(* CODESYS project tc3_component.library
   Company: Zerlauth
   DefaultNamespace: Tc3_Component
   Version: 0.0.0.0
   Author: Peter Zerlauth
   DocFormat: reStructuredText
   Placeholder: Tc3_Component
   Description: ISA88 State Model with Observer and Events
   Title: Tc3_Component

Project tree, tasks and I/O mapping:
  libraries: Tc2_Standard, * (Beckhoff Automation GmbH); Tc2_System, * (Beckhoff Automation GmbH); Tc2_Utilities, * (Beckhoff Automation GmbH)
  Component/
    Event/
      data type E_Error
      data type E_Event
      function block FB_Event [ST]: FB_init, M_Abort, M_AddBOOL, M_AddINT, M_AddREAL, M_AddSTRING, M_AddTIME, M_Arguments, M_Complete, M_Debug, M_Default, M_Error, M_Hold, M_Information, M_Pause, M_Stop, M_Warning, P_Logger
      interface I_Event: M_Abort, M_AddBOOL, M_AddINT, M_AddREAL, M_AddSTRING, M_AddTIME, M_Complete, M_Debug, M_Error, M_Hold, M_Information, M_Pause, M_Stop, M_Warning, P_Logger
      data type ST_Event
      data type ST_EventFlags
    Info/
      function block FB_Info [ST]: FB_init, P_Class, P_Comment, P_Instance, P_Timestamp
      interface I_Info: P_Class, P_Comment, P_Instance, P_Timestamp
    Observer/
      function block FB_Observer [ST]: FB_exit, M_Attach, M_Clear, M_Detach, M_Find, M_Index, M_Notify, P_Length
      interface I_Observer: M_Attach, M_Detach, M_Notify
    Sequence/
      data type E_Sequence
      function block FB_Sequence [ST]: FB_init, M_Await, M_Reset, P_Number
      interface I_Sequence: M_Await, M_Reset, P_Number
    data type E_Mode
    data type E_Request
    data type E_State
    function block FB_Component [ST]: M_Mode, M_Request, M_Aborted, M_Aborting, M_Completed, M_Completing, M_Execute, M_Held, M_Holding, M_Idle, M_Initialise, M_Paused, M_Pausing, M_Resetting, M_Resuming, M_Running, M_Starting, M_Stopped, M_Stopping, M_Unholding, FB_init, M_Cycle, M_OnMode, M_OnNotify, M_OnState, P_Event, P_Identifier, P_Info, P_Mode, P_Observer, P_State
    interface I_Component: M_Cycle, M_Mode, M_OnNotify, M_Request, P_Event, P_Identifier, P_Info, P_Mode, P_Observer, P_State
  List/
    function block FB_ListComponent [ST]: FB_exit, M_Add, M_Clear, M_Find, M_Index, M_Remove, M_Request, P_Length
    function block FB_ListLogger [ST]: FB_exit, M_Add, M_Clear, M_Find, M_Index, M_Remove, P_Length
    function block FB_ListObject [ST]: FB_exit, M_Add, M_Clear, M_Find, M_Index, M_Remove, P_Length
    function block FB_ListString [ST]: FB_exit, M_Add, M_Clear, M_Find, M_Index, M_Remove, P_Length
    interface I_ListComponent: M_Add, M_Clear, M_Find, M_Index, M_Remove, M_Request, P_Length
    interface I_ListLogger: M_Add, M_Clear, M_Find, M_Index, M_Remove, P_Length
    interface I_ListObject: M_Add, M_Clear, M_Find, M_Index, M_Remove, P_Length
    interface I_ListString: M_Add, M_Clear, M_Find, M_Index, M_Remove, P_Length
  Logger/
    function block FB_FileLogger [ST]: M_Log
    function block FB_Logger [ST]: M_Log
    function block FB_TcLogger [ST]: M_Log
  LoggerFactory/
    function block FB_LoggerFactory [ST]: M_Attach, M_Dettach, M_Find, M_Log, M_Publish, M_Remove, M_Reset, M_Start, P_Tags
    interface I_Logger: M_Log
    data type ST_LoggerFactoryTags
  Module/
    function block FB_ModuleBase [ST]: M_Aborted, M_Attach, M_Cycle, M_Dettach, M_Idle, M_Initialise, M_OnMode, M_Resetting, M_Resuming, M_Running, M_Starting, M_Stopped, M_Unholding
    interface I_Module
  Object/
    interface I_Object
  Utils/
    Analog/
      function block AnalogInput [ST]: P_Identifier, P_State, P_Value
      function block AnalogInputREAL [ST]: P_Identifier, P_State, P_Value
      function block AnalogOutput [ST]: FB_init, P_Identifier, P_State, P_Value
      interface I_AnalogChannel: P_Value
    Digital/
      function block FB_DigitalInput [ST]: P_Identifier, P_State, P_Value
      function block FB_DigitalOutput [ST]: P_Identifier, P_State, P_Value
      interface I_Channel: P_Identifier, P_State
      interface I_DigitalChannel: P_Value
    File/
      function block FB_File [ST]: M_Append, M_AppendLine, M_Close, M_Create, M_Delete, M_Load, M_Open, M_Read, M_Write, P_Error
      interface I_File: M_Append, M_AppendLine, M_Close, M_Create, M_Delete, M_Load, M_Open, M_Read, M_Write, P_Error
    function block FB_Debounce [ST]
  global variables Globals
  Klassendiagramm
  global variables Parameters
*)

// Component/Event/E_Error
{attribute 'qualified_only'}
{attribute 'strict'}
{attribute 'to_string'}
TYPE E_Error :
(
	None		:= 0,
    Pause       := 4,	
    Hold      	:= 8,
	Complete	:= 16,	
	Stop		:= 32,
	Abort       := 64
);
END_TYPE

// Component/Event/E_Event
{attribute 'qualified_only'}
{attribute 'strict'}
{attribute 'to_string'}
TYPE E_Event :
(
	Verbose			:= 0,
	Debug			:= 1,
	Information		:= 2,
	Warning			:= 3,
	Error			:= 4
);
END_TYPE

// Component/Event/ST_Event
TYPE ST_Event :
STRUCT
	iSource:		I_Component;
	eEventType:		E_Event;
	nTimestamp:   	ULINT;
	sID:			STRING(10);
	sInstance:		STRING(255);
	sClass:			STRING(255);
	sMessage:		STRING(255);
	sDefault:		STRING(255);
	sArguments:		STRING(255);
	stFlags:		ST_EventFlags;
END_STRUCT
END_TYPE

// Component/Event/ST_EventFlags
TYPE ST_EventFlags :
STRUCT
	bActive:		BIT;
	bRemove:		BIT;
	bPause:			BIT;
	bHold:			BIT;
	bComplete:		BIT;
END_STRUCT
END_TYPE

// Component/Sequence/E_Sequence
{attribute 'qualified_only'}
{attribute 'strict'}
{attribute 'to_string'}
TYPE E_Sequence :
(
	Manual			:= -32768,
	Start			:= 0,
	Done			:= 32767
);
END_TYPE

// Component/E_Mode
{attribute 'qualified_only'}
{attribute 'strict'}
{attribute 'to_string'}
TYPE E_Mode :
(
	{attribute 'hide'}
    Undefined   := 0,
	Automatic   := 1,
    Semiauto    := 2,
	Manual		:= 3
);
END_TYPE

// Component/E_Request
{attribute 'qualified_only'}
{attribute 'strict'}
{attribute 'to_string'}
TYPE E_Request :
(
	{attribute 'hide'}
    Undefined   := 0,
	Reset       := 1,
    Start       := 2,
    Pause       := 4,	
    Hold      	:= 8,
	Complete	:= 16,	
	Stop		:= 32,
	Abort       := 64
);
END_TYPE

// Component/E_State
{attribute 'qualified_only'}
{attribute 'strict'}
{attribute 'to_string'}
TYPE E_State :
(
	{attribute 'hide'}
	Undefined		:= 0,
	Idle			:= 1,
	
// Start
	Starting		:= 2,
	Execute			:= 3,
	
// Pause
	Pausing			:= 4,
	Paused			:= 5,
	Resuming		:= 6,
	
// Hold
	Holding			:= 7,
	Held			:= 8,
	Unholding		:= 9,
	
// Complete
	Completing		:= 10,
	Completed		:= 11,

// Stop
	Stopping		:= 12,
	Stopped			:= 13,

// Abort	
	Aborting		:= 14,
	Aborted			:= 15,

// Reset
	Resetting		:= 16

);
END_TYPE

// LoggerFactory/ST_LoggerFactoryTags
TYPE ST_LoggerFactoryTags :
STRUCT
	bInformation:				BOOL;
	bWarning:					BOOL;
	bError:						BOOL;
	bPause:						BOOL;
	bHold:						BOOL;
	bComplete:					BOOL;	
END_STRUCT
END_TYPE

// Globals
VAR_GLOBAL
	{IF (defined (release))}
    	{attribute 'hide'}
	{END_IF}
	fbLogger:			FB_Logger;
END_VAR

// Parameters
{attribute 'qualified_only'}
VAR_GLOBAL CONSTANT
	nEvents:						INT:= 49;		// Maximum of Events displayed in each Module
END_VAR

// Component/Event/FB_Event
FUNCTION_BLOCK FB_Event IMPLEMENTS I_Event
VAR_INPUT
END_VAR
VAR_OUTPUT
END_VAR
VAR
	fbList:				FB_ListString;
	iParent:			I_Component;
	iLogger:			I_Logger;
	stEvent:			ST_Event;
END_VAR

// https://github.com/PeterZerlauth/Tc3_Component

METHOD FB_init : BOOL
VAR_INPUT
	bInitRetains : BOOL; // if TRUE, the retain variables are initialized (warm start / cold start)
	bInCopyCode : BOOL;  // if TRUE, the instance afterwards gets moved into the copy code (online change)
	iParent:			I_Component;
END_VAR
THIS^.iParent:= iParent;
END_METHOD

METHOD PUBLIC M_Abort
VAR_INPUT
	sMessage:				STRING(255);
	sID:					STRING(10);
END_VAR
stEvent.sMessage:= sMessage;
stEvent.iSource:= iParent;
stEvent.sInstance:= iParent.P_Info.P_Instance;
stEvent.sClass:= iParent.P_Info.P_Class;
stEvent.eEventType:= E_Event.Error;
stEvent.nTimestamp:= F_GetSystemTime();
stEvent.sID:= sID;
stEvent.sDefault:= M_Default(sMessage);
stEvent.sArguments:= M_Arguments();
stEvent.stFlags.bActive:= TRUE;
stEvent.stFlags.bRemove:= FALSE;
stEvent.stFlags.bPause:= FALSE;
stEvent.stFlags.bHold:= FALSE;
stEvent.stFlags.bComplete:= FALSE;

IF iLogger <> 0 THEN
	iLogger.M_Log(stEvent);
ELSE
	fbLogger.M_Log(stEvent);
END_IF

iParent.M_Request(E_Request.Abort);
END_METHOD

METHOD PUBLIC M_AddBOOL
VAR_INPUT
	Value: 	bool;
END_VAR
fbList.M_Add(BOOL_TO_STRING(Value));
END_METHOD

METHOD PUBLIC M_AddINT
VAR_INPUT
	Value: 	LINT;
END_VAR
fbList.M_Add(LINT_TO_STRING(Value));
END_METHOD

METHOD PUBLIC M_AddREAL
VAR_INPUT
	Value: 	Lreal;
	Decimals: INT;
END_VAR
fbList.M_Add(LREAL_TO_FMTSTR(Value, Decimals, TRUE));
END_METHOD

METHOD PUBLIC M_AddSTRING
VAR_INPUT
	Value: STRING(255);
END_VAR
fbList.M_Add(Value);
END_METHOD

METHOD PUBLIC M_AddTIME
VAR_INPUT
	Value: 	TIME;
END_VAR
fbList.M_Add(TIME_TO_STRING(Value));
END_METHOD

METHOD INTERNAL M_Arguments : STRING(255)
VAR_INPUT
END_VAR
VAR
	nIndex:			INT;
END_VAR
WHILE nIndex < fbList. P_Length DO
	M_Arguments:= Concat(Concat(M_Arguments, fbList.M_Index(nIndex)), '$N');
	nIndex:= nIndex + 1;
END_WHILE

fbList.M_Clear();
END_METHOD

METHOD PUBLIC M_Complete
VAR_INPUT
	sMessage:				STRING(255);
	sID:					STRING(10);
END_VAR
stEvent.sMessage:= sMessage;
stEvent.iSource:= iParent;
stEvent.sInstance:= iParent.P_Info.P_Instance;
stEvent.sClass:= iParent.P_Info.P_Class;
stEvent.eEventType:= E_Event.Error;
stEvent.nTimestamp:= F_GetSystemTime();
stEvent.sID:= sID;
stEvent.sDefault:= M_Default(sMessage);
stEvent.sArguments:= M_Arguments();
stEvent.stFlags.bActive:= TRUE;
stEvent.stFlags.bRemove:= FALSE;
stEvent.stFlags.bPause:= FALSE;
stEvent.stFlags.bHold:= False;
stEvent.stFlags.bComplete:= TRUE;

IF iLogger <> 0 THEN
	iLogger.M_Log(stEvent);
ELSE
	iParent.M_Request(E_Request.Complete);
	fbLogger.M_Log(stEvent);
END_IF
END_METHOD

METHOD PUBLIC M_Debug
VAR_INPUT
	Message:				STRING(255);
END_VAR
stEvent.sMessage:= Message;
stEvent.iSource:= iParent;
stEvent.sInstance:= iParent.P_Info.P_Instance;
stEvent.sClass:= iParent.P_Info.P_Class;
stEvent.eEventType:= E_Event.Debug;
stEvent.nTimestamp:= F_GetSystemTime();
stEvent.sID:= '';
stEvent.sDefault:= M_Default(Message);
stEvent.sArguments:= M_Arguments();
stEvent.stFlags.bActive:= TRUE;
stEvent.stFlags.bRemove:= TRUE;
stEvent.stFlags.bPause:= FALSE;
stEvent.stFlags.bHold:= FALSE;
stEvent.stFlags.bComplete:= FALSE;

IF iLogger <> 0 THEN
	iLogger.M_Log(stEvent);
ELSE
	fbLogger.M_Log(stEvent);
END_IF
END_METHOD

METHOD INTERNAL M_Default : STRING(255)
VAR_INPUT
	sMessage:		STRING(255);
END_VAR
VAR
	nIndex:		   	DINT;
	nPosition: 		INT;
END_VAR
nPosition:= Find(sMessage, '%s');
WHILE nPosition <> 0 DO
	sMessage:= Replace(sMessage, fbList.M_Index(nIndex), 2, nPosition);
	nPosition:= Find(sMessage, '%s');
	nIndex:= nIndex + 1;
END_WHILE
M_Default:= sMessage;
END_METHOD

METHOD PUBLIC M_Error
VAR_INPUT
	sMessage:				STRING(255);
	sID:					STRING(10);
END_VAR
stEvent.sMessage:= sMessage;
stEvent.iSource:= iParent;
stEvent.sInstance:= iParent.P_Info.P_Instance;
stEvent.sClass:= iParent.P_Info.P_Class;
stEvent.eEventType:= E_Event.Error;
stEvent.nTimestamp:= F_GetSystemTime();
stEvent.sID:= sID;
stEvent.sDefault:= M_Default(sMessage);
stEvent.sArguments:= M_Arguments();
stEvent.stFlags.bActive:= TRUE;
stEvent.stFlags.bRemove:= TRUE;
stEvent.stFlags.bPause:= FALSE;
stEvent.stFlags.bHold:= FALSE;
stEvent.stFlags.bComplete:= FALSE;

IF iLogger <> 0 THEN
	iLogger.M_Log(stEvent);
ELSE
	fbLogger.M_Log(stEvent);
END_IF
END_METHOD

METHOD PUBLIC M_Hold
VAR_INPUT
	sMessage:				STRING(255);
	sID:					STRING(10);
END_VAR
stEvent.sMessage:= sMessage;
stEvent.iSource:= iParent;
stEvent.sInstance:= iParent.P_Info.P_Instance;
stEvent.sClass:= iParent.P_Info.P_Class;
stEvent.eEventType:= E_Event.Error;
stEvent.nTimestamp:= F_GetSystemTime();
stEvent.sID:= sID;
stEvent.sDefault:= M_Default(sMessage);
stEvent.sArguments:= M_Arguments();
stEvent.stFlags.bActive:= TRUE;
stEvent.stFlags.bRemove:= FALSE;
stEvent.stFlags.bPause:= FALSE;
stEvent.stFlags.bHold:= TRUE;
stEvent.stFlags.bComplete:= FALSE;

IF iLogger <> 0 THEN
	iLogger.M_Log(stEvent);
ELSE
	iParent.M_Request(E_Request.Hold);
	fbLogger.M_Log(stEvent);
END_IF
END_METHOD

METHOD PUBLIC M_Information
VAR_INPUT
	Message:				STRING(255);
	ID:						STRING(10);
END_VAR
stEvent.sMessage:= Message;
stEvent.iSource:= iParent;
stEvent.sInstance:= iParent.P_Info.P_Instance;
stEvent.sClass:= iParent.P_Info.P_Class;
stEvent.eEventType:= E_Event.Information;
stEvent.nTimestamp:= F_GetSystemTime();
stEvent.sID:= ID;
stEvent.sDefault:= M_Default(Message);
stEvent.sArguments:= M_Arguments();
stEvent.stFlags.bActive:= TRUE;
stEvent.stFlags.bRemove:= TRUE;
stEvent.stFlags.bPause:= FALSE;
stEvent.stFlags.bHold:= FALSE;
stEvent.stFlags.bComplete:= FALSE;

IF iLogger <> 0 THEN
	iLogger.M_Log(stEvent);
ELSE
	fbLogger.M_Log(stEvent);
END_IF
END_METHOD

METHOD PUBLIC M_Pause
VAR_INPUT
	sMessage:				STRING(255);
	sID:					STRING(10);
END_VAR
stEvent.sMessage:= sMessage;
stEvent.iSource:= iParent;
stEvent.sInstance:= iParent.P_Info.P_Instance;
stEvent.sClass:= iParent.P_Info.P_Class;
stEvent.eEventType:= E_Event.Error;
stEvent.nTimestamp:= F_GetSystemTime();
stEvent.sID:= sID;
stEvent.sDefault:= M_Default(sMessage);
stEvent.sArguments:= M_Arguments();
stEvent.stFlags.bActive:= TRUE;
stEvent.stFlags.bRemove:= FALSE;
stEvent.stFlags.bPause:= TRUE;
stEvent.stFlags.bHold:= FALSE;
stEvent.stFlags.bComplete:= FALSE;

IF iLogger <> 0 THEN
	iLogger.M_Log(stEvent);
ELSE
	iParent.M_Request(E_Request.Pause);
	fbLogger.M_Log(stEvent);
END_IF
END_METHOD

METHOD PUBLIC M_Stop
VAR_INPUT
	sMessage:				STRING(255);
	sID:					STRING(10);
END_VAR
stEvent.sMessage:= sMessage;
stEvent.iSource:= iParent;
stEvent.sInstance:= iParent.P_Info.P_Instance;
stEvent.sClass:= iParent.P_Info.P_Class;
stEvent.eEventType:= E_Event.Error;
stEvent.nTimestamp:= F_GetSystemTime();
stEvent.sID:= sID;
stEvent.sDefault:= M_Default(sMessage);
stEvent.sArguments:= M_Arguments();
stEvent.stFlags.bActive:= TRUE;
stEvent.stFlags.bRemove:= FALSE;
stEvent.stFlags.bPause:= FALSE;
stEvent.stFlags.bHold:= FALSE;
stEvent.stFlags.bComplete:= FALSE;

IF iLogger <> 0 THEN
	iLogger.M_Log(stEvent);
ELSE
	fbLogger.M_Log(stEvent);
END_IF

iParent.M_Request(E_Request.Stop);
END_METHOD

METHOD PUBLIC M_Warning
VAR_INPUT
	Message:				STRING(255);
	ID:						STRING(10);
END_VAR
stEvent.sMessage:= Message;
stEvent.iSource:= iParent;
stEvent.sInstance:= iParent.P_Info.P_Instance;
stEvent.sClass:= iParent.P_Info.P_Class;
stEvent.eEventType:= E_Event.Warning;
stEvent.nTimestamp:= F_GetSystemTime();
stEvent.sID:= ID;
stEvent.sDefault:= M_Default(Message);
stEvent.sArguments:= M_Arguments();
stEvent.stFlags.bActive:= TRUE;
stEvent.stFlags.bRemove:= TRUE;
stEvent.stFlags.bPause:= FALSE;
stEvent.stFlags.bHold:= FALSE;
stEvent.stFlags.bComplete:= FALSE;

IF iLogger<> 0 THEN
	iLogger.M_Log(stEvent);
ELSE
	fbLogger.M_Log(stEvent);
END_IF
END_METHOD

PROPERTY PUBLIC P_Logger : I_Logger
GET
P_Logger:= iLogger;
END_GET
SET
iLogger:= P_Logger;
END_SET
END_PROPERTY

END_FUNCTION_BLOCK

// Component/Event/I_Event
INTERFACE I_Event EXTENDS I_Object

METHOD PUBLIC M_Abort
VAR_INPUT
	sMessage:				STRING(255);
	sID:					STRING(10);
END_VAR
END_METHOD

METHOD PUBLIC M_AddBOOL
VAR_INPUT
	Value: 	BOOL;
END_VAR
END_METHOD

METHOD PUBLIC M_AddINT
VAR_INPUT
	Value: 	LINT;
END_VAR
END_METHOD

METHOD PUBLIC M_AddREAL
VAR_INPUT
	Value: 	Lreal;
	Decimals: INT;
END_VAR
END_METHOD

METHOD PUBLIC M_AddSTRING
VAR_INPUT
	Value: STRING(255);
END_VAR
END_METHOD

METHOD PUBLIC M_AddTIME
VAR_INPUT
	Value: 	TIME;
END_VAR
END_METHOD

METHOD PUBLIC M_Complete
VAR_INPUT
	sMessage:				STRING(255);
	sID:					STRING(10);
END_VAR
END_METHOD

METHOD PUBLIC M_Debug
VAR_INPUT
	Message:				STRING(255);
END_VAR
END_METHOD

METHOD PUBLIC M_Error
VAR_INPUT
	sMessage:				STRING(255);
	sID:					STRING(10);
END_VAR
END_METHOD

METHOD PUBLIC M_Hold
VAR_INPUT
	sMessage:				STRING(255);
	sID:					STRING(10);
END_VAR
END_METHOD

METHOD PUBLIC M_Information
VAR_INPUT
	Message:				STRING(255);
	ID:						STRING(10);
END_VAR
END_METHOD

METHOD PUBLIC M_Pause
VAR_INPUT
	sMessage:				STRING(255);
	sID:					STRING(10);
END_VAR
END_METHOD

METHOD PUBLIC M_Stop
VAR_INPUT
	sMessage:				STRING(255);
	sID:					STRING(10);
END_VAR
END_METHOD

METHOD PUBLIC M_Warning
VAR_INPUT
	Message:				STRING(255);
	ID:						STRING(10);
END_VAR
END_METHOD

PROPERTY PUBLIC P_Logger : I_Logger
GET
END_GET
SET
END_SET
END_PROPERTY

END_INTERFACE

// Object/I_Object
INTERFACE I_Object EXTENDS __SYSTEM.IQueryInterface

END_INTERFACE

// LoggerFactory/I_Logger
INTERFACE I_Logger EXTENDS I_Object

METHOD PUBLIC M_Log
VAR_INPUT
	stEvent:		ST_Event;
END_VAR
END_METHOD

END_INTERFACE

// List/FB_ListString
{attribute 'no_explicit_call' := 'do not call this POU directly'} 
FUNCTION_BLOCK FB_ListString IMPLEMENTS I_ListString
VAR
	pList: 			POINTER TO STRING(255);
	nLength:		DINT;
	{IF (defined (release))}
    	{attribute 'hide'}
	{END_IF}
	aList:			POINTER TO POINTER TO ARRAY [0..49] OF STRING(255):=ADR(pList);
END_VAR

// https://github.com/PeterZerlauth/Tc3_Component

METHOD FB_exit : BOOL
VAR_INPUT
	bInCopyCode : BOOL; // if TRUE, the exit method is called for exiting an instance that is copied afterwards (online change).
END_VAR
M_Clear();
END_METHOD

METHOD PUBLIC M_Add : BOOL
VAR_INPUT
	Object: 	STRING(255);
END_VAR
VAR
	pOldList: 	POINTER TO STRING(255);
END_VAR
IF Object <> '' THEN
	// First Item
	IF pList = 0 THEN
		nLength:= nLength + 1;
		pList:= __NEW(STRING(255),DINT_TO_UDINT(nLength));
	ELSE
		// Item already in List
		IF M_Find(Object) = -1 THEN
			// backup 
			pOldList:= pList;
			// new Length
			nLength:= nLength + 1;
			// new pointer
			pList:= __NEW(STRING(255),DINT_TO_UDINT(nLength));
			// restore
			Memcpy(pList,pOldList, SIZEOF(STRING(255))*DINT_TO_UDINT(nLength -1));
			// delete old
			__DELETE(pOldList);
		ELSE
			M_Add:= FALSE;	
			RETURN;
		END_IF
	END_IF
	IF pList = 0 THEN
		RETURN;
	END_IF
	// add new Object
	pList[nLength-1]:= Object;
	M_Add:= TRUE;
ELSE
	M_Add:= FALSE;	
END_IF
END_METHOD

METHOD PUBLIC M_Clear : BOOL
IF pList <> 0 THEN
	nLength:= 0;
	__DELETE(pList);
END_IF
M_Clear:= True;
END_METHOD

METHOD PUBLIC M_Find : DINT
VAR_INPUT
	Object: 	STRING(255);
END_VAR
VAR
	nIndex: 	UINT;
END_VAR
// Object already in List
M_Find := -1;
WHILE nIndex < nLength DO
    IF (pList[nIndex] = Object) THEN
        M_Find := nIndex;
        RETURN;
    END_IF
	nIndex := nIndex + 1;
END_WHILE
END_METHOD

METHOD PUBLIC M_Index : STRING(255)
VAR_INPUT
	Index: 	DINT;
END_VAR
IF Index <= nLength THEN
	M_Index:= pList[Index];
ELSE
	M_Index:= '';
END_IF
END_METHOD

METHOD PUBLIC M_Remove : BOOL
VAR_INPUT
	Object: 	STRING(255);
END_VAR
VAR
	pOldList:			POINTER TO STRING(255);
	nPosition: 			DINT;
END_VAR
IF Object <> '' THEN
	// First Item
	IF nLength >= 0 THEN
		// Item already in List
		nPosition:= M_Find(Object);
		IF nPosition <> -1 THEN
			// backup 
			pOldList:= pList;
			// new Length
			nLength:= nLength -1;
			// new pointer
			pList:= __NEW(POINTER TO I_Object,DINT_TO_UDINT(nLength));
			// restore lower part
			Memcpy(pList,pOldList, SIZEOF(STRING(255)) * DINT_TO_UDINT(nPosition));
			//pList[nPosition]:= iObject;
			Memcpy(pList + (SIZEOF(STRING(255))*nPosition),pOldList + (SIZEOF(STRING(255))*(nPosition + 1)), SIZEOF(STRING(255)) * DINT_TO_UDINT(nLength - nPosition));
			// delete old
			__DELETE(pOldList);
		ELSE
			M_Remove:= FALSE;	
			RETURN;
		END_IF
	ELSE
		M_Remove:= FALSE;	
		RETURN;
	END_IF
	M_Remove:= TRUE;
ELSE
	M_Remove:= FALSE;	
END_IF
END_METHOD

PROPERTY PUBLIC P_Length : DINT
GET
P_Length:= nLength;
END_GET
END_PROPERTY

END_FUNCTION_BLOCK

// List/I_ListString
INTERFACE I_ListString EXTENDS I_Object

METHOD PUBLIC M_Add : BOOL
VAR_INPUT
	Object: 	STRING(255);
END_VAR
END_METHOD

METHOD PUBLIC M_Clear : BOOL
END_METHOD

METHOD PUBLIC M_Find : DINT
VAR_INPUT
	Object: 	STRING(255);
END_VAR
END_METHOD

METHOD PUBLIC M_Index : STRING(255)
VAR_INPUT
	Index: 	DINT;
END_VAR
END_METHOD

METHOD PUBLIC M_Remove : BOOL
VAR_INPUT
	Object: 	STRING(255);
END_VAR
END_METHOD

PROPERTY PUBLIC P_Length : DINT
GET
END_GET
END_PROPERTY

END_INTERFACE

// Component/I_Component
INTERFACE I_Component EXTENDS I_Object

METHOD PUBLIC M_Cycle
VAR_INPUT
END_VAR
END_METHOD

METHOD PUBLIC M_Mode : BOOL
VAR_INPUT
	eMode:		E_Mode;
END_VAR
END_METHOD

METHOD PUBLIC M_OnNotify
VAR_INPUT
	eRequest:					E_Request;
	eMode:						E_Mode;
END_VAR
END_METHOD

METHOD PUBLIC M_Request : BOOL
VAR_INPUT
	eRequest:	E_Request;
END_VAR
END_METHOD

PROPERTY PUBLIC P_Event : I_Event
GET
END_GET
END_PROPERTY

PROPERTY PUBLIC P_Identifier : STRING(25)
GET
END_GET
SET
END_SET
END_PROPERTY

PROPERTY PUBLIC P_Info : I_Info
GET
END_GET
END_PROPERTY

PROPERTY PUBLIC P_Mode : E_Mode
GET
END_GET
END_PROPERTY

PROPERTY PUBLIC P_Observer : I_Observer
GET
END_GET
END_PROPERTY

PROPERTY PUBLIC P_State : E_State
GET
END_GET
END_PROPERTY

END_INTERFACE

// Component/Info/I_Info
INTERFACE I_Info EXTENDS I_Object

PROPERTY PUBLIC P_Class : String(255)
GET
END_GET
END_PROPERTY

PROPERTY PUBLIC P_Comment : String(255)
GET
END_GET
END_PROPERTY

PROPERTY PUBLIC P_Instance : String(255)
GET
END_GET
END_PROPERTY

PROPERTY PUBLIC P_Timestamp : ULINT
GET
END_GET
END_PROPERTY

END_INTERFACE

// Component/Observer/I_Observer
INTERFACE I_Observer

METHOD M_Attach : BOOL
VAR_INPUT
	Object: 	I_Component;
END_VAR
END_METHOD

METHOD M_Detach : BOOL
VAR_INPUT
	Object: 	I_Component;
END_VAR
END_METHOD

METHOD M_Notify : BOOL
VAR_INPUT
	eRequest:					E_Request;
	eMode:						E_Mode;
END_VAR
END_METHOD

END_INTERFACE

// Component/Info/FB_Info
FUNCTION_BLOCK PUBLIC FB_Info IMPLEMENTS I_Info
VAR_INPUT
	sIdentifier:						STRING(25);					// Identifier
END_VAR
VAR_OUTPUT
END_VAR
VAR
    sInstancePath:				REFERENCE TO STRING(255);
	fbReadSymInfo: 				PLC_ReadSymInfoByNameEx;
END_VAR
VAR_STAT
	nCycle: 					UDINT;
	nTimestamp: 				ULINT;
END_VAR

// https://github.com/PeterZerlauth/Tc3_Component
IF nCycle <> TwinCAT_SystemInfoVarList._TaskInfo[GETCURTASKINDEXEX()].CycleCount THEN
	nCycle:= TwinCAT_SystemInfoVarList._TaskInfo[GETCURTASKINDEXEX()].CycleCount;
	nTimestamp:= F_GetSystemTime();
END_IF

fbReadSymInfo(
	NETID:= , 
	PORT:= , 
	SYMNAME:= , 
	START:= , 
	TMOUT:= , 
	BUSY=> , 
	ERR=> , 
	ERRID=> , 
	SYMINFO=> , 
	OVTYPE=> , 
	OVCOMMENT=> );

METHOD FB_init : BOOL
VAR_INPUT
	bInitRetains : BOOL; // if TRUE, the retain variables are initialized (warm start / cold start)
	bInCopyCode : BOOL;  // if TRUE, the instance afterwards gets moved into the copy code (online change)
	sInstancePath:			REFERENCE TO STRING(255);
END_VAR
VAR
    sName:				STRING(255);
    nPosition:			INT;
END_VAR
THIS^.sInstancePath REF= sInstancePath;

sName := CONCAT(TwinCAT_SystemInfoVarList._AppInfo.ProjectName, '.');

nPosition := FIND(sInstancePath, sName);
IF nPosition > 0 THEN
    fbReadSymInfo.SYMNAME:= DELETE(sInstancePath, nPosition-1 + LEN(sName), 1);
END_IF

nPosition := FIND(fbReadSymInfo.SYMNAME, sName);

IF nPosition > 0 THEN
    fbReadSymInfo.SYMNAME:= DELETE(fbReadSymInfo.SYMNAME, nPosition - 1 + LEN(sName), 1);
END_IF

fbReadSymInfo.PORT:= TwinCAT_SystemInfoVarList._AppInfo.AdsPort;
fbReadSymInfo.START:= TRUE;
END_METHOD

PROPERTY PUBLIC P_Class : String(255)
GET
P_Class:= fbReadSymInfo.SYMINFO.symDataType;
END_GET
END_PROPERTY

PROPERTY PUBLIC P_Comment : String(255)
GET
P_Comment:= fbReadSymInfo.SYMINFO.symComment;
END_GET
END_PROPERTY

PROPERTY PUBLIC P_Instance : String(255)
GET
P_Instance:= fbReadSymInfo.SYMNAME;
END_GET
END_PROPERTY

PROPERTY PUBLIC P_Timestamp : ULINT
GET
P_Timestamp:= nTimestamp;
END_GET
END_PROPERTY

END_FUNCTION_BLOCK

// Component/Observer/FB_Observer
{attribute 'no_explicit_call'} 
FUNCTION_BLOCK PUBLIC FB_Observer IMPLEMENTS I_Observer
VAR
	pList: 			POINTER TO I_Component;
	nLength:		DINT;
	{attribute 'conditionalshow'}
	aList:			POINTER TO POINTER TO ARRAY [0..100] OF I_Component:=ADR(pList);
END_VAR

// https://github.com/PeterZerlauth/Tc3_Component

METHOD FB_exit : BOOL
VAR_INPUT
	bInCopyCode : BOOL; // if TRUE, the exit method is called for exiting an instance that is copied afterwards (online change).
END_VAR
M_Clear();
END_METHOD

METHOD M_Attach : BOOL
VAR_INPUT
	Object: 	I_Component;
END_VAR
VAR
	pOldList: 	POINTER TO I_Component;
END_VAR
IF Object <> 0 THEN
	// First Item
	IF pList = 0 THEN
		nLength:= nLength + 1;
		pList:= __NEW(POINTER TO I_Component,DINT_TO_UDINT(nLength));
	ELSE
		// Item already in List
		IF M_Find(Object) = -1 THEN
			// backup 
			pOldList:= pList;
			// new Length
			nLength:= nLength + 1;
			// new pointer
			pList:= __NEW(POINTER TO I_Component,DINT_TO_UDINT(nLength));
			// restore
			Memcpy(pList,pOldList, SIZEOF(POINTER TO I_Component)*DINT_TO_UDINT(nLength -1));
			// delete old
			__DELETE(pOldList);
		ELSE
			M_Attach:= FALSE;	
			RETURN;
		END_IF
	END_IF
	IF pList = 0 THEN
		RETURN;
	END_IF
	// add new Object
	pList[nLength-1]:= Object;
	M_Attach:= TRUE;
ELSE
	M_Attach:= FALSE;	
END_IF
END_METHOD

METHOD M_Clear
IF pList <> 0 THEN
	nLength:= 0;
	__DELETE(pList);
END_IF
END_METHOD

METHOD M_Detach : BOOL
VAR_INPUT
	Object: 	I_Component;
END_VAR
VAR
	pOldList:			POINTER TO I_Component;
	nPosition: 			DINT;
END_VAR
IF Object <> 0 THEN
	// First Item
	IF nLength >= 0 THEN
		// Item already in List
		nPosition:= M_Find(Object);
		IF nPosition <> -1 THEN
			// backup 
			pOldList:= pList;
			// new Length
			nLength:= nLength -1;
			// new pointer
			pList:= __NEW(POINTER TO I_Component,DINT_TO_UDINT(nLength));
			// restore lower part
			Memcpy(pList,pOldList, SIZEOF(POINTER TO I_Component) * DINT_TO_UDINT(nPosition));
			//pList[nPosition]:= iObject;
			Memcpy(pList + (SIZEOF(POINTER TO I_Component)*nPosition),pOldList + (SIZEOF(POINTER TO I_Component)*(nPosition + 1)), SIZEOF(POINTER TO I_Component) * DINT_TO_UDINT(nLength - nPosition));
			// delete old
			__DELETE(pOldList);
		ELSE
			M_Detach:= FALSE;	
			RETURN;
		END_IF
	ELSE
		M_Detach:= FALSE;	
		RETURN;
	END_IF
	M_Detach:= TRUE;
ELSE
	M_Detach:= FALSE;	
END_IF
END_METHOD

METHOD M_Find : DINT
VAR_INPUT
	Object: 	I_Component;
END_VAR
VAR
	nIndex: 	UINT;
END_VAR
// Object already in List
M_Find := -1;
WHILE nIndex < nLength DO
    IF (pList[nIndex] = Object) THEN
        M_Find := nIndex;
        RETURN;
    END_IF
	nIndex := nIndex + 1;
END_WHILE
END_METHOD

METHOD M_Index : I_Component
VAR_INPUT
	Index: 	DINT;
END_VAR
IF Index <= nLength THEN
	M_Index:= pList[Index];
END_IF
END_METHOD

METHOD M_Notify : BOOL
VAR_INPUT
	eRequest:					E_Request;
	eMode:						E_Mode;
END_VAR

VAR
	nIndex: 	INT;
END_VAR
WHILE nIndex < nLength DO
	pList[nIndex].M_OnNotify(eRequest, eMode);
	nIndex:= nIndex + 1; 
END_WHILE
END_METHOD

PROPERTY P_Length : DINT
GET
P_Length:= nLength;
END_GET
END_PROPERTY

END_FUNCTION_BLOCK

// Component/Sequence/FB_Sequence
FUNCTION_BLOCK FB_Sequence IMPLEMENTS I_Sequence
VAR_INPUT
END_VAR
VAR_OUTPUT
	sMessage:				STRING(255);
	nNumber:				INT;
END_VAR
VAR
	iParent:			I_Component;
	fbTimeout:			TON;
	fbDelay: 			TON;
END_VAR

// https://github.com/PeterZerlauth/Tc3_Component
IF iParent.P_Mode = E_Mode.Manual THEN
	nNumber:= E_Sequence.Manual;
END_IF

METHOD FB_init : BOOL
VAR_INPUT
	bInitRetains : BOOL; // if TRUE, the retain variables are initialized (warm start / cold start)
	bInCopyCode : BOOL;  // if TRUE, the instance afterwards gets moved into the copy code (online change)
	iParent:			I_Component;
END_VAR
THIS^.iParent:= iParent;
END_METHOD

METHOD PUBLIC M_Await 
VAR_INPUT
	sMessage:				STRING(255);		
	tTimeout:				TIME;
	tDelay:					TIME;	
	bPause:					BOOL;
	bReturn:				BOOL;
	nNumber:				INT;
END_VAR
THIS^.sMessage:= sMessage;
IF bReturn THEN
	IF tDelay <> T#0S THEN
		fbDelay(IN:= TRUE);
		IF fbDelay.Q THEN
			THIS^.nNumber:= nNumber;
			fbDelay(IN:= FALSE);
			IF bPause THEN
				IF iParent.P_Mode = E_Mode.Semiauto THEN
					iParent.M_Request(E_Request.Pause);		
				END_IF
			END_IF	
		END_IF
	ELSE
		THIS^.nNumber:= nNumber;
		fbTimeout(IN:= FALSE);
		IF bPause THEN
			IF iParent.P_Mode = E_Mode.Semiauto THEN
				iParent.M_Request(E_Request.Pause);		
			END_IF
		END_IF	
	END_IF		
ELSE
	IF tTimeout <> T#0S THEN
		fbTimeout(IN:= TRUE);
		IF fbTimeout.Q THEN
			iParent.P_Event.M_AddINT(THIS^.nNumber);
			iParent.P_Event.M_Stop('Timeout in sequence number %s', '');
		END_IF
	END_IF
END_IF
END_METHOD

METHOD M_Reset
nNumber:= E_Sequence.Start;
fbDelay(IN:= FALSE);
fbTimeout(IN:= FALSE);
END_METHOD

PROPERTY PUBLIC P_Number : int
GET
P_Number:= nNumber;
END_GET
SET
nNumber:= P_Number;
END_SET
END_PROPERTY

END_FUNCTION_BLOCK

// Component/Sequence/I_Sequence
INTERFACE I_Sequence EXTENDS I_Object

METHOD PUBLIC M_Await 
VAR_INPUT
	sMessage:				STRING(255);
	tTimeout:				TIME;
	tDelay:					TIME;	
	bPause:					BOOL;
	bReturn:				BOOL;
	nNumber:				INT;
END_VAR
END_METHOD

METHOD M_Reset
END_METHOD

PROPERTY PUBLIC P_Number : int
GET
END_GET
SET
END_SET
END_PROPERTY

END_INTERFACE

// Component/FB_Component
{attribute 'reflection'} 
{attribute 'no_explicit_call' := 'do not call this POU directly'} 
FUNCTION_BLOCK FB_Component IMPLEMENTS I_Component
VAR_INPUT
END_VAR
VAR_OUTPUT
END_VAR
VAR
    {attribute 'hide'}
	{attribute 'instance-path'} 
    {attribute 'noinit'}
    sInstancePath:					STRING(255);				// Instance-Path
	fbInfo:							FB_Info(sInstancePath);		// Info about function block
	fbObserver:						FB_Observer;				// Observer
	fbEvent:						FB_Event(THIS^);			// Event creator
	fbSequence:						FB_Sequence(THIS^);			// Sequence (abort = reset)
	eStateRequest:					E_Request;					// State command
	{attribute 'OPC.UA.DA' := '1'}
	{ attribute 'TcHmiSymbol' }
	eState:							E_State;					// Current state
    {attribute 'hide'}
	eStatePrevious:					E_State;					// Previous state
	eModeRequest:					E_Mode;						// Requested mode
	{attribute 'OPC.UA.DA' := '1'}
	{attribute 'TcHmiSymbol' }
	eMode:							E_Mode;						// Current mode
    {attribute 'hide'}
	eModePrevious:					E_Mode;						// Previous mode	
END_VAR

// https://github.com/PeterZerlauth/Tc3_Component

METHOD PUBLIC M_Mode : BOOL
VAR_INPUT
	eMode:		E_Mode;
END_VAR
IF eMode = E_Mode.Undefined THEN
	M_Mode:= TRUE;
ELSE
	IF THIS^.eMode = eMode THEN
		M_Mode:= TRUE;
	ELSE
		eModeRequest:= eMode;	
	END_IF	
END_IF
END_METHOD

METHOD PUBLIC M_Request : BOOL
VAR_INPUT
	eRequest:	E_Request;
END_VAR
// Request component states / Command Pattern
CASE eRequest OF
	E_Request.Undefined:
		M_Request:= TRUE;
		
	E_Request.Start:
		IF eState = E_State.Execute THEN
			M_Request:= TRUE;
		ELSE
			eStateRequest:= eRequest;				
		END_IF
		
	E_Request.Pause:
		IF eState >= E_State.Paused THEN
			M_Request:= TRUE;
		ELSE
			IF eStateRequest < eRequest THEN
				eStateRequest:= eRequest;				
			END_IF		
		END_IF
		
	E_Request.Hold:
		IF eState >= E_State.Held THEN
			M_Request:= TRUE;
		ELSE
			IF eStateRequest < eRequest THEN
				eStateRequest:= eRequest;				
			END_IF		
		END_IF
		
	E_Request.Complete:
		IF eState = E_State.Completed THEN
			M_Request:= TRUE;
		ELSE
			IF eStateRequest < eRequest THEN
				eStateRequest:= eRequest;				
			END_IF		
		END_IF
		
	E_Request.Stop:
		IF eState = E_State.Stopped THEN
			M_Request:= TRUE;
		ELSE
			IF eStateRequest < eRequest THEN
				eStateRequest:= eRequest;				
			END_IF		
		END_IF
		
	E_Request.Abort:
		IF eState = E_State.Aborted THEN
			M_Request:= TRUE;
		ELSE
			IF eStateRequest < eRequest THEN
				eStateRequest:= eRequest;				
			END_IF		
		END_IF

	E_Request.Reset:
		IF eState = E_State.Idle THEN
			M_Request:= TRUE;
		ELSE
			eStateRequest:= eRequest;			
		END_IF
END_CASE
END_METHOD

METHOD PROTECTED M_Aborted
VAR_INPUT
END_VAR
END_METHOD

METHOD PROTECTED M_Aborting : BOOL // Return state complete
VAR_INPUT
END_VAR
// State Aborting
M_Aborting:= TRUE;
END_METHOD

METHOD PROTECTED M_Completed
VAR_INPUT
END_VAR
END_METHOD

METHOD PROTECTED M_Completing : BOOL // Return state complete
VAR_INPUT
END_VAR
// State Completing
M_Completing:= True;
END_METHOD

METHOD PROTECTED M_Execute : BOOL // Return state complete
VAR_INPUT
END_VAR
M_Execute:= True;
END_METHOD

METHOD PROTECTED M_Held
VAR_INPUT
END_VAR
END_METHOD

METHOD PROTECTED M_Holding : BOOL // Return state complete
VAR_INPUT
END_VAR
// State Holding
M_Holding:= True;
END_METHOD

METHOD PROTECTED M_Idle
VAR_INPUT
END_VAR
// State Idle
END_METHOD

METHOD PROTECTED M_Initialise
VAR_INPUT
END_VAR
END_METHOD

METHOD PROTECTED M_Paused // Return state complete
VAR_INPUT
END_VAR
END_METHOD

METHOD PROTECTED M_Pausing : BOOL
VAR_INPUT
END_VAR
// State Holding
M_Pausing:= True;
END_METHOD

METHOD PROTECTED M_Resetting : BOOL // Return state complete
VAR_INPUT
END_VAR
// State Resetting
M_Resetting:= True;
END_METHOD

METHOD PROTECTED M_Resuming : BOOL // Return state complete
VAR_INPUT
END_VAR
// State Holding
M_Resuming:= True;
END_METHOD

METHOD PROTECTED M_Running
VAR_INPUT
END_VAR
// Will be called in all running states, for monitorings which not only in one state active
END_METHOD

METHOD PROTECTED M_Starting : BOOL // Return state complete
VAR_INPUT
END_VAR
// State Starting
M_Starting:= True;
END_METHOD

METHOD PROTECTED M_Stopped
VAR_INPUT
END_VAR
END_METHOD

METHOD PROTECTED M_Stopping : BOOL // Return state complete
VAR_INPUT
END_VAR
// State Stopping
M_Stopping:= True;
END_METHOD

METHOD PROTECTED M_Unholding : BOOL // Return state complete
VAR_INPUT
END_VAR
// State Holding
M_Unholding:= True;
END_METHOD

METHOD FB_init : BOOL
VAR_INPUT
	bInitRetains : BOOL; // if TRUE, the retain variables are initialized (warm start / cold start)
	bInCopyCode : BOOL:= TRUE;
END_VAR
M_Initialise();
END_METHOD

METHOD PUBLIC M_Cycle
VAR_INPUT
END_VAR
fbInfo();
fbObserver();
fbEvent();
fbSequence();

// Handle Module Type Package states
CASE eState OF
	E_State.Undefined:
		M_Initialise();
		eMode:= E_Mode.Automatic;
		eState:= E_State.Idle;					
		
	E_State.Resetting:
		M_Running();
		IF M_Resetting() THEN
			eState:= E_State.Idle;
			eStateRequest:= E_Request.Undefined;
		END_IF
		CASE eStateRequest OF
			E_Request.Stop:
				eState:= E_State.Stopping;
				
			E_Request.Abort:
				eState:= E_State.Aborting;
				
		END_CASE
		
	E_State.Idle:
		M_Running();
		M_Idle();
		CASE eStateRequest OF
			
			E_Request.Start:
				eState:= E_State.Starting;
				
			E_Request.Stop:
				eState:= E_State.Stopping;
				
			E_Request.Abort:
				eState:= E_State.Aborting;
				
			ELSE
				eStateRequest:= E_Request.Undefined;
				
		END_CASE

	E_State.Starting:
		M_Running();
		IF M_Starting() THEN
			eState:= E_State.Execute;
			eStateRequest:= E_Request.Undefined;
		END_IF
		CASE eStateRequest OF
			
			E_Request.Stop:
				eState:= E_State.Stopping;
				
			E_Request.Abort:
				eState:= E_State.Aborting;
				
		END_CASE

	E_State.Execute:
		M_Running();
		IF M_Execute() THEN
			CASE eStateRequest OF
				
				E_Request.Complete:
					eState:= E_State.Completing;
					
			END_CASE
		END_IF
		CASE eStateRequest OF
			E_Request.Complete:;
			E_Request.Stop:
				eState:= E_State.Stopping;
				
			E_Request.Abort:
				eState:= E_State.Aborting;

			E_Request.Hold:
				eState:= E_State.Holding;
				
			E_Request.Pause:
				eState:= E_State.Pausing;
				
			ELSE
				eStateRequest:= E_Request.Undefined;
				
		END_CASE
		
	E_State.Stopping:
		M_Running();
		IF M_Stopping() THEN
			eState:= E_State.Stopped;
			eStateRequest:= E_Request.Undefined;
		END_IF
		CASE eStateRequest OF
			
			E_Request.Abort:
				eState:= E_State.Aborting;
				
		END_CASE

	E_State.Stopped:
		M_Stopped();
		CASE eStateRequest OF
			
			E_Request.Abort:
				eState:= E_State.Aborting;
				
			E_Request.Reset:
				eState:= E_State.Resetting;
				
		ELSE
			eStateRequest:= E_Request.Undefined;				
		END_CASE
		
		
	E_State.Aborting:
		fbSequence.M_Reset();
		IF M_Aborting() THEN
			eState:= E_State.Aborted;
			eStateRequest:= E_Request.Undefined;
		END_IF
		
	E_State.Aborted:
		M_Aborted();
		CASE eStateRequest OF
			
			E_Request.Reset:
				eState:= E_State.Resetting;
				
		ELSE
			eStateRequest:= E_Request.Undefined;				
		END_CASE

		
	E_State.Pausing:
		M_Running();
		IF M_Pausing() THEN
			eState:= E_State.Paused;
			eStateRequest:= E_Request.Undefined;
		END_IF
		CASE eStateRequest OF
			
			E_Request.Stop:
				eState:= E_State.Stopping;
				
			E_Request.Abort:
				eState:= E_State.Aborting;

		END_CASE
		
	
	E_State.Paused:
		M_Running();
		M_Paused();
		CASE eStateRequest OF
			
			E_Request.Start:
				eState:= E_State.Resuming;
				
			E_Request.Stop:
				eState:= E_State.Stopping;
				
			E_Request.Abort:
				eState:= E_State.Aborting;
						
		ELSE
			eStateRequest:= E_Request.Undefined;

		END_CASE
		
	E_State.Resuming:
		M_Running();
		IF M_Resuming() THEN
			eState:= E_State.Execute;
		END_IF
		CASE eStateRequest OF
			
			E_Request.Stop:
				eState:= E_State.Stopping;
				
			E_Request.Abort:
				eState:= E_State.Aborting;

		END_CASE

	E_State.Holding:
		M_Running();
		IF M_Holding() THEN
			eState:= E_State.Held;
			eStateRequest:= E_Request.Undefined;
		END_IF
		CASE eStateRequest OF
			
			E_Request.Stop:
				eState:= E_State.Stopping;
				
			E_Request.Abort:
				eState:= E_State.Aborting;

		END_CASE

	E_State.Held:
		M_Running();
		M_Held();
		CASE eStateRequest OF
			
			E_Request.Start:
				eState:= E_State.Unholding;

			E_Request.Stop:
				eState:= E_State.Stopping;
				
			E_Request.Abort:
				eState:= E_State.Aborting;
				
			ELSE
				eStateRequest:= E_Request.Undefined;

		END_CASE
		
	E_State.Unholding:
		M_Running();
		IF M_Unholding() THEN
			eState:= E_State.Execute;
		END_IF
		CASE eStateRequest OF
			
			E_Request.Stop:
				eState:= E_State.Stopping;
				
			E_Request.Abort:
				eState:= E_State.Aborting;

		END_CASE
		
	E_State.Completing:
		M_Running();
		IF M_Completing() THEN
			eState:= E_State.Completed;
			eStateRequest:= E_Request.Undefined;
		END_IF
		CASE eStateRequest OF
			
			E_Request.Stop:
				eState:= E_State.Stopping;
				
			E_Request.Abort:
				eState:= E_State.Aborting;

		END_CASE
		
	E_State.Completed:
		M_Running();
		M_Completed();
		CASE eStateRequest OF
			
			E_Request.Stop:
				eState:= E_State.Stopping;
				
			E_Request.Abort:
				eState:= E_State.Aborting;
					
			E_Request.Reset:
				eState:= E_State.Resetting;
				
			ELSE
				eStateRequest:= E_Request.Undefined;
				
		END_CASE
		
END_CASE

IF eModeRequest <> E_Mode.Undefined THEN
	IF 	eMode <> eModeRequest THEN
		eMode:= eModeRequest;
		fbObserver.M_Notify(0, eMode);		
	END_IF
END_IF
eModeRequest:= E_Mode.Undefined;

// Detect mode changed
IF eModePrevious <> eMode THEN
	M_OnMode(eMode, eModePrevious);
	eModePrevious:= eMode;
END_IF
	
// Detect state changed
IF eStatePrevious <> eState THEN
	M_OnState(eState, eStatePrevious);
	eStatePrevious:= eState;
END_IF

CASE eStateRequest of
	E_Request.Undefined, E_Request.Start, E_Request.Pause, E_Request.Hold:
		// Ignore
	ELSE
		fbObserver.M_Notify(eStateRequest, 0);
END_CASE
END_METHOD

METHOD PROTECTED M_OnMode
VAR_INPUT
	eMode:							E_Mode;						// Current mode
	eModePrevious:					E_Mode;						// Previous mode	
END_VAR
END_METHOD

METHOD PUBLIC M_OnNotify
VAR_INPUT
	eRequest:					E_Request;
	eMode:						E_Mode;
END_VAR
// Method will be called by the Observer
M_Request(eRequest);
M_Mode(eMode);
END_METHOD

METHOD Protected M_OnState
VAR_INPUT
	eState:							E_State;						// Current state
	eStatePrevious:					E_State;						// Previous state	
END_VAR
END_METHOD

PROPERTY PUBLIC P_Event : I_Event
GET
P_Event:= fbEvent;
END_GET
END_PROPERTY

PROPERTY PUBLIC P_Identifier : STRING(25)
GET
P_Identifier:= fbInfo.sIdentifier;
END_GET
SET
PUBLIC 
VAR
END_VAR
fbInfo.sIdentifier:= P_Identifier;
END_SET
END_PROPERTY

PROPERTY PUBLIC P_Info : I_Info
GET
P_Info:= fbInfo;
END_GET
END_PROPERTY

PROPERTY PUBLIC P_Mode : E_Mode
GET
P_Mode:= eMode;
END_GET
END_PROPERTY

PROPERTY PUBLIC P_Observer : I_Observer
GET
P_Observer:= fbObserver;
END_GET
END_PROPERTY

PROPERTY PUBLIC P_State : E_State
GET
P_State:= eState;
END_GET
END_PROPERTY

END_FUNCTION_BLOCK

// List/FB_ListComponent
{attribute 'no_explicit_call' := 'do not call this POU directly'} 
FUNCTION_BLOCK FB_ListComponent IMPLEMENTS I_ListComponent
VAR
	nLength:		DINT;
	pList: 			POINTER TO I_Component;
	{IF (defined (release))}
    	{attribute 'hide'}
	{END_IF}
	aList:			POINTER TO POINTER TO ARRAY [0..49] OF I_Component:=ADR(pList);
END_VAR

// https://github.com/PeterZerlauth/Tc3_Component

METHOD FB_exit : BOOL
VAR_INPUT
	bInCopyCode : BOOL; // if TRUE, the exit method is called for exiting an instance that is copied afterwards (online change).
END_VAR
M_Clear();
END_METHOD

METHOD PUBLIC M_Add : BOOL
VAR_INPUT
	Object: 	I_Component;
END_VAR
VAR
	pOldList: 	POINTER TO I_Component;
END_VAR
IF Object <> 0 THEN
	// First Item
	IF pList = 0 THEN
		nLength:= nLength + 1;
		pList:= __NEW(POINTER TO I_Component,DINT_TO_UDINT(nLength));
	ELSE
		// Item already in List
		IF M_Find(Object) = -1 THEN
			// backup 
			pOldList:= pList;
			// new Length
			nLength:= nLength + 1;
			// new pointer
			pList:= __NEW(POINTER TO I_Component,DINT_TO_UDINT(nLength));
			// restore
			Memcpy(pList,pOldList, SIZEOF(POINTER TO I_Component)*DINT_TO_UDINT(nLength -1));
			// delete old
			__DELETE(pOldList);
		ELSE
			M_Add:= FALSE;	
			RETURN;
		END_IF
	END_IF
	IF pList = 0 THEN
		RETURN;
	END_IF
	// add new Object
	pList[nLength-1]:= Object;
	M_Add:= TRUE;
ELSE
	M_Add:= FALSE;	
END_IF
END_METHOD

METHOD PUBLIC M_Clear : BOOL
// Clear
IF pList <> 0 THEN
	nLength:= 0;
	__DELETE(pList);
END_IF
M_Clear:= TRUE;
END_METHOD

METHOD PUBLIC M_Find : DINT
VAR_INPUT
	Object: 	I_Component;
END_VAR
VAR
	nIndex: 	UINT;
END_VAR
// Find
M_Find := -1;
WHILE nIndex < nLength DO
    IF (pList[nIndex] = Object) THEN
        M_Find := nIndex;
        RETURN;
    END_IF
	nIndex := nIndex + 1;
END_WHILE
END_METHOD

METHOD PUBLIC M_Index : I_Component
VAR_INPUT
	Index: 	DINT;
END_VAR
// Index
IF Index <= nLength THEN
	M_Index:= pList[Index];
END_IF
END_METHOD

METHOD PUBLIC M_Remove : BOOL
VAR_INPUT
	Object: 	I_Component;
END_VAR
VAR
	pOldList:			POINTER TO I_Component;
	nPosition: 			DINT;
END_VAR
// Remove
IF Object <> 0 THEN
	// First Item
	IF nLength >= 0 THEN
		// Item already in List
		nPosition:= M_Find(Object);
		IF nPosition <> -1 THEN
			// backup 
			pOldList:= pList;
			// new Length
			nLength:= nLength -1;
			// new pointer
			pList:= __NEW(POINTER TO I_Component,DINT_TO_UDINT(nLength));
			// restore lower part
			Memcpy(pList,pOldList, SIZEOF(POINTER TO I_Object) * DINT_TO_UDINT(nPosition));
			//pList[nPosition]:= iObject;
			Memcpy(pList + (SIZEOF(POINTER TO I_Component)*nPosition),pOldList + (SIZEOF(POINTER TO I_Component)*(nPosition + 1)), SIZEOF(POINTER TO I_Component) * DINT_TO_UDINT(nLength - nPosition));
			// delete old
			__DELETE(pOldList);
		ELSE
			M_Remove:= FALSE;	
			RETURN;
		END_IF
	ELSE
		M_Remove:= FALSE;	
		RETURN;
	END_IF
	M_Remove:= TRUE;
ELSE
	M_Remove:= FALSE;	
END_IF
END_METHOD

METHOD PUBLIC M_Request : BOOL
VAR_INPUT
	eRequest:		E_Request;
END_VAR

VAR
	nIndex: 		INT;
END_VAR
M_Request:= TRUE;
WHILE nIndex < nLength DO
	M_Request:= M_Request AND M_Index(nIndex).M_Request(eRequest);
	nIndex:= nIndex +1;
END_WHILE
END_METHOD

PROPERTY PUBLIC P_Length : DINT
GET
P_Length:= nLength;
END_GET
END_PROPERTY

END_FUNCTION_BLOCK

// List/I_ListComponent
INTERFACE I_ListComponent

METHOD PUBLIC M_Add : BOOL
VAR_INPUT
	Object: 	I_Component;
END_VAR
END_METHOD

METHOD PUBLIC M_Clear : BOOL
END_METHOD

METHOD PUBLIC M_Find : DINT
VAR_INPUT
	Object: 	I_Component;
END_VAR
END_METHOD

METHOD PUBLIC M_Index : I_Component
VAR_INPUT
	Index: 	DINT;
END_VAR
END_METHOD

METHOD PUBLIC M_Remove : BOOL
VAR_INPUT
	Object: 	I_Component;
END_VAR
END_METHOD

METHOD PUBLIC M_Request : BOOL
VAR_INPUT
	eRequest:	E_Request;
END_VAR
END_METHOD

PROPERTY P_Length : DINT
GET
END_GET
END_PROPERTY

END_INTERFACE

// List/FB_ListLogger
{attribute 'no_explicit_call' := 'do not call this POU directly'} 
FUNCTION_BLOCK FB_ListLogger IMPLEMENTS I_ListLogger
VAR
	nLength:		DINT;
	pList: 			POINTER TO I_Logger;
	{IF (defined (release))}
    	{attribute 'hide'}
	{END_IF}
	aList:			POINTER TO POINTER TO ARRAY [0..49] OF I_Logger:=ADR(pList);
END_VAR

// https://github.com/PeterZerlauth/Tc3_Component

METHOD FB_exit : BOOL
VAR_INPUT
	bInCopyCode : BOOL; // if TRUE, the exit method is called for exiting an instance that is copied afterwards (online change).
END_VAR
M_Clear();
END_METHOD

METHOD PUBLIC M_Add : BOOL
VAR_INPUT
	Object: 	I_Logger;
END_VAR
VAR
	pOldList: 	POINTER TO I_Logger;
END_VAR
IF Object <> 0 THEN
	// First Item
	IF pList = 0 THEN
		nLength:= nLength + 1;
		pList:= __NEW(POINTER TO I_Logger,DINT_TO_UDINT(nLength));
	ELSE
		// Item already in List
		IF M_Find(Object) = -1 THEN
			// backup 
			pOldList:= pList;
			// new Length
			nLength:= nLength + 1;
			// new pointer
			pList:= __NEW(POINTER TO I_Logger,DINT_TO_UDINT(nLength));
			// restore
			Memcpy(pList,pOldList, SIZEOF(POINTER TO I_Logger)*DINT_TO_UDINT(nLength -1));
			// delete old
			__DELETE(pOldList);
		ELSE
			M_Add:= FALSE;	
			RETURN;
		END_IF
	END_IF
	IF pList = 0 THEN
		RETURN;
	END_IF
	// add new Object
	pList[nLength-1]:= Object;
	M_Add:= TRUE;
ELSE
	M_Add:= FALSE;	
END_IF
END_METHOD

METHOD PUBLIC M_Clear : bool
IF pList <> 0 THEN
	nLength:= 0;
	__DELETE(pList);
END_IF
M_Clear:= True;
END_METHOD

METHOD PUBLIC M_Find : DINT
VAR_INPUT
	Object: 	I_Logger;
END_VAR
VAR
	nIndex: 	UINT;
END_VAR
// Object already in List
M_Find := -1;
WHILE nIndex < nLength DO
    IF (pList[nIndex] = Object) THEN
        M_Find := nIndex;
        RETURN;
    END_IF
	nIndex := nIndex + 1;
END_WHILE
END_METHOD

METHOD PUBLIC M_Index : I_Logger
VAR_INPUT
	Index: 	DINT;
END_VAR
IF Index <= nLength THEN
	M_Index:= pList[Index];
END_IF
END_METHOD

METHOD PUBLIC M_Remove : BOOL
VAR_INPUT
	Object: 	I_Logger;
END_VAR
VAR
	pOldList:			POINTER TO I_Logger;
	nPosition: 			DINT;
END_VAR
IF Object <> 0 THEN
	// First Item
	IF nLength >= 0 THEN
		// Item already in List
		nPosition:= M_Find(Object);
		IF nPosition <> -1 THEN
			// backup 
			pOldList:= pList;
			// new Length
			nLength:= nLength -1;
			// new pointer
			pList:= __NEW(POINTER TO I_Object,DINT_TO_UDINT(nLength));
			// restore lower part
			Memcpy(pList,pOldList, SIZEOF(POINTER TO I_Logger) * DINT_TO_UDINT(nPosition));
			//pList[nPosition]:= iObject;
			Memcpy(pList + (SIZEOF(POINTER TO I_Logger)*nPosition),pOldList + (SIZEOF(POINTER TO I_Logger)*(nPosition + 1)), SIZEOF(POINTER TO I_Logger) * DINT_TO_UDINT(nLength - nPosition));
			// delete old
			__DELETE(pOldList);
		ELSE
			M_Remove:= FALSE;	
			RETURN;
		END_IF
	ELSE
		M_Remove:= FALSE;	
		RETURN;
	END_IF
	M_Remove:= TRUE;
ELSE
	M_Remove:= FALSE;	
END_IF
END_METHOD

PROPERTY PUBLIC P_Length : DINT
GET
P_Length:= nLength;
END_GET
END_PROPERTY

END_FUNCTION_BLOCK

// List/I_ListLogger
INTERFACE I_ListLogger

METHOD PUBLIC M_Add : BOOL
VAR_INPUT
	Object: 	I_Logger;
END_VAR
END_METHOD

METHOD PUBLIC M_Clear : BOOL
END_METHOD

METHOD PUBLIC M_Find : DINT
VAR_INPUT
	Object: 	I_Logger;
END_VAR
END_METHOD

METHOD PUBLIC M_Index : I_Logger
VAR_INPUT
	Index: 	DINT;
END_VAR
END_METHOD

METHOD PUBLIC M_Remove : BOOL
VAR_INPUT
	Object: 	I_Logger;
END_VAR
END_METHOD

PROPERTY P_Length : DINT
GET
END_GET
END_PROPERTY

END_INTERFACE

// List/FB_ListObject
{attribute 'no_explicit_call' := 'do not call this POU directly'} 
FUNCTION_BLOCK FB_ListObject IMPLEMENTS I_ListObject
VAR
	nLength:		DINT;
	pList: 			POINTER TO I_Object;
	{IF (defined (release))}
    	{attribute 'hide'}
	{END_IF}
	aList:			POINTER TO POINTER TO ARRAY [0..49] OF I_Object:=ADR(pList);
END_VAR

// https://github.com/PeterZerlauth/Tc3_Component

METHOD FB_exit : BOOL
VAR_INPUT
	bInCopyCode : BOOL; // if TRUE, the exit method is called for exiting an instance that is copied afterwards (online change).
END_VAR
M_Clear();
END_METHOD

METHOD PUBLIC M_Add : BOOL
VAR_INPUT
	Object: 	I_Object;
END_VAR
VAR
	pOldList: 	POINTER TO I_Object;
END_VAR
IF Object <> 0 THEN
	// First Item
	IF pList = 0 THEN
		nLength:= nLength + 1;
		pList:= __NEW(POINTER TO I_Object,DINT_TO_UDINT(nLength));
	ELSE
		// Item already in List
		IF M_Find(Object) = -1 THEN
			// backup 
			pOldList:= pList;
			// new Length
			nLength:= nLength + 1;
			// new pointer
			pList:= __NEW(POINTER TO I_Object,DINT_TO_UDINT(nLength));
			// restore
			Memcpy(pList,pOldList, SIZEOF(POINTER TO I_Object)*DINT_TO_UDINT(nLength -1));
			// delete old
			__DELETE(pOldList);
		ELSE
			M_Add:= FALSE;	
			RETURN;
		END_IF
	END_IF
	IF pList = 0 THEN
		RETURN;
	END_IF
	// add new Object
	pList[nLength-1]:= Object;
	M_Add:= TRUE;
ELSE
	M_Add:= FALSE;	
END_IF
END_METHOD

METHOD PUBLIC M_Clear : bool
IF pList <> 0 THEN
	nLength:= 0;
	__DELETE(pList);
END_IF
M_Clear:= True;
END_METHOD

METHOD PUBLIC M_Find : DINT
VAR_INPUT
	Object: 	I_Object;
END_VAR
VAR
	nIndex: 	UINT;
END_VAR
// Object already in List
M_Find := -1;
WHILE nIndex < nLength DO
    IF (pList[nIndex] = Object) THEN
        M_Find := nIndex;
        RETURN;
    END_IF
	nIndex := nIndex + 1;
END_WHILE
END_METHOD

METHOD PUBLIC M_Index : I_Object
VAR_INPUT
	Index: 	DINT;
END_VAR
IF Index <= nLength THEN
	M_Index:= pList[Index];
END_IF
END_METHOD

METHOD PUBLIC M_Remove : BOOL
VAR_INPUT
	Object: 	I_Object;
END_VAR
VAR
	pOldList:			POINTER TO I_Object;
	nPosition: 			DINT;
END_VAR
IF Object <> 0 THEN
	// First Item
	IF nLength >= 0 THEN
		// Item already in List
		nPosition:= M_Find(Object);
		IF nPosition <> -1 THEN
			// backup 
			pOldList:= pList;
			// new Length
			nLength:= nLength -1;
			// new pointer
			pList:= __NEW(POINTER TO I_Object,DINT_TO_UDINT(nLength));
			// restore lower part
			Memcpy(pList,pOldList, SIZEOF(POINTER TO I_Object) * DINT_TO_UDINT(nPosition));
			//pList[nPosition]:= iObject;
			Memcpy(pList + (SIZEOF(POINTER TO I_Object)*nPosition),pOldList + (SIZEOF(POINTER TO I_Object)*(nPosition + 1)), SIZEOF(POINTER TO I_Object) * DINT_TO_UDINT(nLength - nPosition));
			// delete old
			__DELETE(pOldList);
		ELSE
			M_Remove:= FALSE;	
			RETURN;
		END_IF
	ELSE
		M_Remove:= FALSE;	
		RETURN;
	END_IF
	M_Remove:= TRUE;
ELSE
	M_Remove:= FALSE;	
END_IF
END_METHOD

PROPERTY PUBLIC P_Length : DINT
GET
P_Length:= nLength;
END_GET
END_PROPERTY

END_FUNCTION_BLOCK

// List/I_ListObject
INTERFACE I_ListObject

METHOD PUBLIC M_Add : BOOL
VAR_INPUT
	Object: 	I_Object;
END_VAR
END_METHOD

METHOD PUBLIC M_Clear : BOOL
END_METHOD

METHOD PUBLIC M_Find : DINT
VAR_INPUT
	Object: 	I_Object;
END_VAR
END_METHOD

METHOD PUBLIC M_Index : I_Object
VAR_INPUT
	Index: 	DINT;
END_VAR
END_METHOD

METHOD PUBLIC M_Remove : BOOL
VAR_INPUT
	Object: 	I_Object;
END_VAR
END_METHOD

PROPERTY P_Length : DINT
GET
END_GET
END_PROPERTY

END_INTERFACE

// Logger/FB_FileLogger
FUNCTION_BLOCK FB_FileLogger IMPLEMENTS I_Logger
VAR
	fbFile:					FB_File;
END_VAR

// https://github.com/PeterZerlauth/Tc3_Component

METHOD M_Log
VAR_INPUT
	stEvent	: 		ST_Event;
END_VAR

VAR
	sMessage:			STRING(255);
END_VAR
sMessage:= Concat(Concat(stEvent.sInstance, ' | '), stEvent.sDefault);
END_METHOD

END_FUNCTION_BLOCK

// Utils/File/FB_File
{attribute 'no_explicit_call'} 
FUNCTION_BLOCK FB_File
VAR
    fbCreateDir:	FB_CreateDir;
	fbOpen:			FB_FileOpen;
	fbRead:			FB_FileRead;
	fbLoad:			FB_FileLoad;
	fbWrite:		FB_FileWrite;
	fbClose:		FB_FileClose;
	fbDelete:		FB_FileDelete;
END_VAR
VAR_OUTPUT
	nError:			UDINT;
END_VAR

// https://github.com/PeterZerlauth/Tc3_Component

METHOD PUBLIC M_Append : BOOL
VAR_INPUT
	Text:			STRING(255);
END_VAR
fbWrite();
IF fbWrite.bExecute THEN
	IF fbWrite.bError THEN
		nError:= fbWrite.nErrId;
		fbWrite.bExecute:= FALSE;
	ELSIF fbWrite.bBusy THEN
		;
	ELSE
		M_Append:= TRUE;
		fbWrite.bExecute:= FALSE;
	END_IF
ELSE
	fbWrite.bExecute:= TRUE;
	fbWrite.pWriteBuff:= ADR(Text);
	fbWrite.cbWriteLen:= INT_TO_UDINT(Len(Text));
END_IF
END_METHOD

METHOD PUBLIC M_AppendLine : BOOL
VAR_INPUT
	Text:			STRING(255);
END_VAR
Text:= Concat(Text, '$R');
M_AppendLine:= M_Append(Text);
END_METHOD

METHOD PUBLIC M_Close : BOOL
VAR_INPUT
END_VAR
fbClose();
IF fbClose.bExecute THEN
	IF fbClose.hFile = 0 THEN
		fbClose.bExecute:= FALSE;
		M_Close:= TRUE;
	ELSIF fbClose.bError THEN
		fbClose.bExecute:= FALSE;
		nError:= fbClose.nErrId;
	ELSIF fbClose.bBusy THEN
		;
	ELSE
		nError:= 0;	
		fbRead.hFile:= 0;
		fbWrite.hFile:= 0;
		fbClose.hFile:= 0;
		fbClose.bExecute:= FALSE;
		M_Close:= TRUE;
	END_IF
ELSE
	fbClose.bExecute:= TRUE;
END_IF
END_METHOD

METHOD PUBLIC M_Create : BOOL
VAR_INPUT
	PathName:		STRING(255);
END_VAR
VAR
	nTemp: INT;
END_VAR
VAR_INST
	nPosition: INT;
END_VAR
fbCreateDir();
nTemp := FIND(RIGHT(PathName, LEN(PathName) - nPosition), '\');
if nTemp <> 0 then
	IF fbCreateDir.bExecute THEN
		IF NOT fbCreateDir.bBusy THEN
			nPosition := nPosition + nTemp;
			fbCreateDir.bExecute:= FALSE;
		END_IF
	ELSE
		fbCreateDir.bExecute:= TRUE;
		fbCreateDir.ePath:= PATH_GENERIC;
		fbCreateDir.sPathName:= Left(PathName, nPosition + nTemp);
	END_IF
ELSE
	IF M_Open(PathName) THEN
		M_Create:= TRUE;
		nPosition:= 0;
	END_IF
END_IF
END_METHOD

METHOD PUBLIC M_Delete : BOOL
VAR_INPUT
	PathName:		STRING(255);
END_VAR
fbDelete();
IF fbDelete.bExecute THEN
	IF fbDelete.bError THEN
		fbDelete.bExecute:= FALSE;
		M_Delete:= TRUE;
	ELSIF fbDelete.bBusy THEN
		;
	ELSE
		fbDelete.bExecute:= FALSE;
		M_Delete:= TRUE;
	END_IF
ELSE
	fbDelete.bExecute:= TRUE;
	fbDelete.sPathName:= PathName;
	fbDelete.ePath:= E_OpenPath.PATH_GENERIC;
END_IF
END_METHOD

METHOD PUBLIC M_Load : BOOL
VAR_INPUT
	PathName:		STRING(255);
	Value:			ANY;
END_VAR
fbLoad();
IF fbLoad.bExecute THEN
	IF fbLoad.bError THEN
		nError:= fbLoad.nErrId;
		fbLoad.bExecute:= FALSE;
	ELSIF fbLoad.bBusy THEN
		;
	ELSE
		M_Load:= TRUE;
	END_IF
ELSE
	fbLoad.sPathName:= PathName;
	fbLoad.bExecute:= TRUE;
	fbLoad.pReadBuff:= Value.pValue;
	fbLoad.cbReadLen:= DINT_TO_UDINT(Value.diSize);
END_IF
END_METHOD

METHOD PUBLIC M_Open : BOOL
VAR_INPUT
	PathName:		STRING(255);
END_VAR
fbOpen();
IF fbOpen.bExecute THEN
	IF fbOpen.bError THEN
		nError:= fbOpen.nErrId;
		fbOpen.bExecute:= FALSE;
	ELSIF fbOpen.bBusy THEN
		;
	ELSE
		fbRead.hFile:= fbOpen.hFile;
		fbWrite.hFile:= fbOpen.hFile;
		fbClose.hFile:= fbOpen.hFile;
		fbOpen.bExecute:= FALSE;
		M_Open:= TRUE;
	END_IF	
ELSE
	fbOpen.bExecute:= TRUE;
	fbOpen.sPathName:= PathName;
	fbOpen.nMode:= (FOPEN_MODEAPPEND OR FOPEN_MODEPLUS OR FOPEN_MODETEXT);
END_IF
END_METHOD

METHOD PUBLIC M_Read : BOOL
VAR_INPUT
	Value:		ANY;
END_VAR
fbRead();
IF fbRead.bExecute THEN
	IF fbRead.bError THEN
		nError:= fbRead.nErrId;
		fbRead.bExecute:= FALSE;
	ELSIF fbRead.bBusy THEN
		;
	ELSE
		fbRead.bExecute:= FALSE;
		M_Read:= TRUE;
	END_IF
ELSE
	fbRead.bExecute:= TRUE;
	fbRead.pReadBuff:= Value.pValue;
	fbRead.cbReadLen:= DINT_TO_UDINT(Value.diSize);
END_IF
END_METHOD

METHOD PUBLIC M_Write : BOOL
VAR_INPUT
	Value:		ANY;
END_VAR
fbWrite();
IF fbWrite.bExecute THEN
	IF fbWrite.bError THEN
		nError:= fbWrite.nErrId;
		fbWrite.bExecute:= FALSE;
	ELSIF fbWrite.bBusy THEN
		M_Write:= FALSE;
	ELSE
		M_Write:= TRUE;
		fbWrite.bExecute:= FALSE;
	END_IF
ELSE
	fbWrite.bExecute:= TRUE;
	fbRead.pReadBuff:= Value.pValue;
	fbRead.cbReadLen:= DINT_TO_UDINT(Value.diSize);
END_IF
END_METHOD

PROPERTY PUBLIC P_Error : UDINT
GET
P_Error:= nError;
END_GET
END_PROPERTY

END_FUNCTION_BLOCK

// Logger/FB_Logger
FUNCTION_BLOCK FB_Logger EXTENDS FB_TcLogger
VAR
END_VAR

// https://github.com/PeterZerlauth/Tc3_Component

METHOD M_Log
VAR_INPUT
	stEvent	: 		ST_Event;
END_VAR

VAR
	sMessage:			STRING(255);
END_VAR
sMessage:= Concat(Concat(stEvent.sInstance, ' | iLogger = 0 | '), stEvent.sDefault);
CASE stEvent.eEventType OF
	E_Event.Error:
		ADSLOGSTR( msgCtrlMask := ADSLOG_MSGTYPE_ERROR , msgFmtStr := '%s', strArg := sMessage);
	E_Event.Warning:
		ADSLOGSTR( msgCtrlMask := ADSLOG_MSGTYPE_WARN , msgFmtStr := '%s', strArg := sMessage);
	E_Event.Information:
		ADSLOGSTR( msgCtrlMask := ADSLOG_MSGTYPE_HINT , msgFmtStr := '%s', strArg := sMessage);
	E_Event.Debug:
		ADSLOGSTR( msgCtrlMask := ADSLOG_MSGTYPE_HINT, msgFmtStr := '%s', strArg := sMessage);
	E_Event.Verbose:
		ADSLOGSTR( msgCtrlMask := ADSLOG_MSGTYPE_HINT , msgFmtStr := '%s', strArg := sMessage);
END_CASE
END_METHOD

END_FUNCTION_BLOCK

// Logger/FB_TcLogger
FUNCTION_BLOCK FB_TcLogger IMPLEMENTS I_Logger
VAR
END_VAR

// https://github.com/PeterZerlauth/Tc3_Component

METHOD M_Log
VAR_INPUT
	stEvent	: 		ST_Event;
END_VAR

VAR
	sMessage:			STRING(255);
END_VAR
sMessage:= Concat(Concat(stEvent.sInstance, ' | '), stEvent.sDefault);
CASE stEvent.eEventType OF
	E_Event.Error:
		ADSLOGSTR( msgCtrlMask := ADSLOG_MSGTYPE_ERROR , msgFmtStr := '%s', strArg := sMessage);
	E_Event.Warning:
		ADSLOGSTR( msgCtrlMask := ADSLOG_MSGTYPE_WARN , msgFmtStr := '%s', strArg := sMessage);
	E_Event.Information:
		ADSLOGSTR( msgCtrlMask := ADSLOG_MSGTYPE_HINT , msgFmtStr := '%s', strArg := sMessage);
	E_Event.Debug:
		ADSLOGSTR( msgCtrlMask := ADSLOG_MSGTYPE_HINT, msgFmtStr := '%s', strArg := sMessage);
	E_Event.Verbose:
		ADSLOGSTR( msgCtrlMask := ADSLOG_MSGTYPE_HINT , msgFmtStr := '%s', strArg := sMessage);
END_CASE
END_METHOD

END_FUNCTION_BLOCK

// LoggerFactory/FB_LoggerFactory
FUNCTION_BLOCK FB_LoggerFactory IMPLEMENTS I_Logger
VAR
	fbList:						FB_ListLogger;
	nLength:					DINT;
	aEvent:						ARRAY [0..Parameters.nEvents] OF ST_Event;	
	nIndex: 					DINT;
	stTags:						ST_LoggerFactoryTags;
END_VAR

// https://github.com/PeterZerlauth/Tc3_Component

// Deactivate old events
stTags.bInformation:= FALSE;
stTags.bWarning:= FALSE;
stTags.bError:= FALSE;
stTags.bPause:= FALSE;
stTags.bHold:= FALSE;
stTags.bComplete:= FALSE;

nIndex:= 0;
WHILE nIndex < nLength DO
	stTags.bPause S= aEvent[nIndex].stFlags.bPause;
	stTags.bHold S= aEvent[nIndex].stFlags.bHold;
	stTags.bComplete S= aEvent[nIndex].stFlags.bComplete;
	CASE aEvent[nIndex].eEventType OF
		E_Event.Error:
			stTags.bError:= TRUE;
		E_Event.Warning:
			stTags.bWarning:= TRUE;	
		E_Event.Information:
			stTags.bInformation:= TRUE;
	END_CASE

	IF aEvent[nIndex].stFlags.bActive THEN
		IF aEvent[nIndex].stFlags.bRemove THEN
			aEvent[nIndex].stFlags.bActive:= FALSE;
		END_IF
	ELSE
		M_Remove(nIndex);
	END_IF
	nIndex := nIndex + 1;
END_WHILE

METHOD PUBLIC M_Attach
VAR_INPUT
	Logger:		I_Logger;
END_VAR
// Attach
fbList.M_Add(Logger);
END_METHOD

METHOD PUBLIC M_Dettach
VAR_INPUT
	Logger:		I_Logger;
END_VAR
// Dettach
fbList.M_Remove(Logger);
END_METHOD

METHOD PUBLIC M_Find : DINT
VAR_INPUT
	stEvent:	ST_Event;
END_VAR
VAR 
	nIndex:		DINT;
END_VAR
// Find event in buffer
M_Find := -1;
WHILE nIndex < nLength DO
	IF (aEvent[nIndex].iSource = stEvent.iSource) AND_THEN
    	(aEvent[nIndex].eEventType = stEvent.eEventType) AND_THEN
		(aEvent[nIndex].sInstance = stEvent.sInstance) AND_THEN
		(aEvent[nIndex].sClass = stEvent.sClass) AND_THEN
		(aEvent[nIndex].sMessage = stEvent.sMessage) THEN
        M_Find := nIndex;
        RETURN;
    END_IF
	nIndex := nIndex + 1;
END_WHILE
END_METHOD

METHOD PUBLIC M_Log
VAR_INPUT
	stEvent:		ST_Event;
END_VAR
VAR
	nIndex:			DINT;
END_VAR
IF (nIndex:=  M_Find(stEvent)) >= 0 THEN
	// Update existing events
	aEvent[nIndex].sArguments:= stEvent.sArguments;
	aEvent[nIndex].sDefault:= stEvent.sDefault;
	aEvent[nIndex].stFlags:= stEvent.stFlags;
ELSE
	// add new event
	aEvent[nLength].stFlags:= stEvent.stFlags;
	aEvent[nLength]:= stEvent;
	nLength:= nLength + 1;
	// Publish to Subscribers
	M_Publish(stEvent);
END_IF
END_METHOD

METHOD M_Publish
VAR_INPUT
	stEvent:	ST_Event;
END_VAR
VAR 
	nIndex:		DINT;
END_VAR
// Publis event
WHILE nIndex < fbList.P_Length DO
	fbList.M_Index(nIndex).M_Log(stEvent);
	nIndex := nIndex + 1;
END_WHILE
END_METHOD

METHOD PUBLIC M_Remove : Bool
VAR_INPUT
	Index:		DINT;
END_VAR
// Remove event
MEMCPY(ADR(aEvent[Index]), ADR(aEvent[Index + 1]), SIZEOF(ST_Event) * DINT_TO_UDINT(Parameters.nEvents - nLength));
nLength:= nLength - 1;
END_METHOD

METHOD PUBLIC M_Reset
VAR_INPUT
END_VAR
// Reset all events
nLength:= 0;
Memset(ADR(aEvent), 0, SIZEOF(aEvent));
END_METHOD

METHOD PUBLIC M_Start
VAR_INPUT
END_VAR
VAR 
	nIndex:		DINT;
END_VAR
nIndex:= 0;
WHILE nIndex < nLength DO
	aEvent[nIndex].stFlags.bHold:= FALSE;
	aEvent[nIndex].stFlags.bPause:= FALSE;	
	nIndex := nIndex + 1;
END_WHILE
END_METHOD

PROPERTY PUBLIC P_Tags : REFERENCE TO ST_LoggerFactoryTags
GET
P_Tags ref= stTags;
END_GET
END_PROPERTY

END_FUNCTION_BLOCK

// Module/FB_ModuleBase
FUNCTION_BLOCK FB_ModuleBase EXTENDS FB_Component
VAR_INPUT
END_VAR
VAR_OUTPUT
END_VAR
VAR
	fbMembers:					FB_ListComponent;
	fbLoggerFactory:			FB_LoggerFactory;;
	fbTcLogger:					FB_TcLogger;
	fbFileLogger:				FB_FileLogger;
END_VAR

// https://github.com/PeterZerlauth/Tc3_Component

METHOD PROTECTED M_Aborted
VAR_INPUT
END_VAR
SUPER^.M_Aborted();
fbEvent.M_AddSTRING(P_Identifier);
fbEvent.M_Information('Module %s aborted, reset', '');
END_METHOD

METHOD PUBLIC M_Attach
VAR_INPUT
	Component:		I_Component;
END_VAR
Component.P_Event.P_Logger:= fbLoggerFactory;
fbMembers.M_Add(Component);
Component.P_Observer.M_Attach(THIS^);
fbObserver.M_Attach(Component);
END_METHOD

METHOD PUBLIC M_Cycle
VAR_INPUT
END_VAR
fbLoggerFactory();

IF fbLoggerFactory.P_Tags.bHold THEN
	M_Request(E_Request.Hold);
ELSIF fbLoggerFactory.P_Tags.bPause THEN
	M_Request(E_Request.Pause);
ELSIF fbLoggerFactory.P_Tags.bComplete THEN
	M_Request(E_Request.Complete);
END_IF

SUPER^.M_Cycle();
END_METHOD

METHOD PUBLIC M_Dettach
VAR_INPUT
	Component:		I_Component;
END_VAR
Component.P_Event.P_Logger:= 0;
fbMembers.M_Remove(Component);
Component.P_Observer.M_Detach(THIS^);
fbObserver.M_Detach(Component);
END_METHOD

METHOD PROTECTED M_Idle
VAR_INPUT
END_VAR
SUPER^.M_Idle();
fbEvent.M_AddSTRING(P_Identifier);
fbEvent.M_Information('Module %s not started', '');
END_METHOD

METHOD PROTECTED M_Initialise
VAR_INPUT
END_VAR
SUPER^.M_Initialise();

fbEvent.P_Logger:= fbLoggerFactory;
fbLoggerFactory.M_Attach(fbTcLogger);
fbLoggerFactory.M_Attach(fbFileLogger);
END_METHOD

METHOD Protected M_OnMode
VAR_INPUT
	eMode:							E_Mode;						// Current mode
	eModePrevious:					E_Mode;						// Previous mode	
END_VAR
CASE eMode OF
	E_Mode.Semiauto, E_Mode.Automatic:
		IF eModePrevious = E_Mode.Manual THEN
			fbEvent.M_AddSTRING(P_Identifier);
			fbEvent.M_Abort('Module %s was in manual mode', '');
		END_IF
END_CASE
END_METHOD

METHOD PROTECTED M_Resetting : BOOL
VAR_INPUT
END_VAR
M_Resetting:= SUPER^.M_Resetting();
fbMembers.M_Request(E_Request.Reset);
fbLoggerFactory.M_Reset();
END_METHOD

METHOD PROTECTED M_Resuming : BOOL // Return state complete
VAR_INPUT
END_VAR
M_Resuming:= fbMembers.M_Request(E_Request.Start);
fbLoggerFactory.M_Start();
END_METHOD

METHOD PROTECTED M_Running
VAR_INPUT
END_VAR
END_METHOD

METHOD PROTECTED M_Starting : BOOL
VAR_INPUT
END_VAR
M_Starting:= fbMembers.M_Request(E_Request.Start);
END_METHOD

METHOD PROTECTED M_Stopped
VAR_INPUT
END_VAR
SUPER^.M_Stopped();
fbEvent.M_AddSTRING(P_Identifier);
fbEvent.M_Information('Module %s stopped, reset', '');
END_METHOD

METHOD PROTECTED M_Unholding : BOOL // Return state complete
VAR_INPUT
END_VAR
M_Unholding:= fbMembers.M_Request(E_Request.Start);
fbLoggerFactory.M_Start();
END_METHOD

END_FUNCTION_BLOCK

// Module/I_Module
INTERFACE I_Module EXTENDS I_Component

END_INTERFACE

// Utils/Analog/AnalogInput
{attribute 'reflection'} 
FUNCTION_BLOCK AnalogInput IMPLEMENTS I_AnalogChannel
VAR_INPUT
END_VAR
VAR_OUTPUT
END_VAR
VAR
	sIdentifier:				STRING(25);	// Equipment ID
	Channel			AT%I*: INT;	// Link to input
END_VAR

// https://github.com/PeterZerlauth/Tc3_Component

PROPERTY PUBLIC P_Identifier : String(25)
GET
P_Identifier:= sIdentifier;
END_GET
END_PROPERTY

PROPERTY P_State : EPlcMappingStatus
GET
P_State:= F_GetMappingStatus(ADR(Channel), SIZEOF(INT));
END_GET
END_PROPERTY

PROPERTY PUBLIC P_Value : Lreal
GET
P_Value:= INT_TO_LREAL(Channel);
END_GET
SET
PUBLIC 
VAR
END_VAR
Channel:= LREAL_TO_INT(P_Value);
END_SET
END_PROPERTY

END_FUNCTION_BLOCK

// Utils/Analog/I_AnalogChannel
INTERFACE I_AnalogChannel EXTENDS I_Channel

PROPERTY P_Value : LREAL
GET
END_GET
SET
END_SET
END_PROPERTY

END_INTERFACE

// Utils/Digital/I_Channel
INTERFACE I_Channel EXTENDS I_Object

PROPERTY PUBLIC P_Identifier : String(25)
GET
END_GET
END_PROPERTY

PROPERTY P_State : EPlcMappingStatus
GET
END_GET
END_PROPERTY

END_INTERFACE

// Utils/Analog/AnalogInputREAL
{attribute 'reflection'} 
FUNCTION_BLOCK AnalogInputREAL IMPLEMENTS I_AnalogChannel
VAR_INPUT
END_VAR
VAR_OUTPUT
END_VAR
VAR
	sIdentifier:				STRING(25);	// Equipment ID
	Channel			AT%I*: REAL;	// Link to input
END_VAR

// https://github.com/PeterZerlauth/Tc3_Component

PROPERTY PUBLIC P_Identifier : String(25)
GET
P_Identifier:= sIdentifier;
END_GET
END_PROPERTY

PROPERTY P_State : EPlcMappingStatus
GET
P_State:= F_GetMappingStatus(ADR(Channel), SIZEOF(INT));
END_GET
END_PROPERTY

PROPERTY PUBLIC P_Value : Lreal
GET
P_Value:= Channel;
END_GET
SET
PUBLIC 
VAR
END_VAR
Channel:= LREAL_TO_INT(P_Value);
END_SET
END_PROPERTY

END_FUNCTION_BLOCK

// Utils/Analog/AnalogOutput
{attribute 'reflection'} 
FUNCTION_BLOCK AnalogOutput IMPLEMENTS I_AnalogChannel
VAR_INPUT
END_VAR
VAR_OUTPUT
END_VAR
VAR
	sIdentifier:				STRING(25);	// Equipment ID
	Channel			AT%Q*: INT;	// Link to input
END_VAR

// https://github.com/PeterZerlauth/Tc3_Component

METHOD FB_init : BOOL
VAR_INPUT
	bInitRetains : BOOL; // if TRUE, the retain variables are initialized (warm start / cold start)
	bInCopyCode : BOOL;  // if TRUE, the instance afterwards gets moved into the copy code (online change)
	ID:				STRING(25);
END_VAR
THIS^.sIdentifier:= ID;
END_METHOD

PROPERTY PUBLIC P_Identifier : String(25)
GET
P_Identifier:= sIdentifier;
END_GET
END_PROPERTY

PROPERTY P_State : EPlcMappingStatus
GET
P_State:= F_GetMappingStatus(ADR(Channel), SIZEOF(INT));
END_GET
END_PROPERTY

PROPERTY PUBLIC P_Value : Lreal
GET
P_Value:= INT_TO_LREAL(Channel);
END_GET
SET
PUBLIC 
VAR
END_VAR
Channel:= LREAL_TO_INT(P_Value);
END_SET
END_PROPERTY

END_FUNCTION_BLOCK

// Utils/Digital/FB_DigitalInput
{attribute 'reflection'} 
FUNCTION_BLOCK FB_DigitalInput IMPLEMENTS I_DigitalChannel
VAR_INPUT
	tDebounce:			TIME:= T#50MS;
END_VAR
VAR_OUTPUT
END_VAR
VAR

	sIdentifier:				STRING(25);	// Equipment ID
	Channel			AT%I*: BOOL;	// Link to input
	fbDebounce:		FB_Debounce;
END_VAR

// https://github.com/PeterZerlauth/Tc3_Component
fbDebounce(bInput:= Channel, tTime:= tDebounce);

PROPERTY PUBLIC P_Identifier : String(25)
GET
P_Identifier:= sIdentifier;
END_GET
END_PROPERTY

PROPERTY P_State : EPlcMappingStatus
GET
P_State:= F_GetMappingStatus(ADR(Channel), SIZEOF(BOOL));
END_GET
END_PROPERTY

PROPERTY PUBLIC P_Value : bool
GET
P_Value:= fbDebounce.bValue;
END_GET
SET
PUBLIC 
VAR
END_VAR
END_SET
END_PROPERTY

END_FUNCTION_BLOCK

// Utils/Digital/I_DigitalChannel
INTERFACE I_DigitalChannel EXTENDS I_Channel

PROPERTY P_Value : bool
GET
END_GET
SET
END_SET
END_PROPERTY

END_INTERFACE

// Utils/FB_Debounce
FUNCTION_BLOCK FB_Debounce 
VAR_INPUT
	bInput:				BOOL;
	tTime:				TIME;
END_VAR
VAR_OUTPUT
	bValue:				BOOL;
END_VAR
VAR
	fbTimerOn:			Ton;
	fbTimerOff:			Ton;
END_VAR

// https://github.com/PeterZerlauth/Tc3_Component
IF bInput THEN
	fbTimerOn(IN:= TRUE, PT:= tTime);
	fbTimerOff(IN:= FALSE);
	IF fbTimerOn.Q THEN
		bValue:= TRUE;
	END_IF
ELSE
	fbTimerOff(IN:= TRUE, PT:= tTime);
	fbTimerOn(IN:= FALSE);
	IF fbTimerOff.Q THEN
		bValue:= FALSE;
	END_IF	
END_IF

END_FUNCTION_BLOCK

// Utils/Digital/FB_DigitalOutput
{attribute 'reflection'} 
FUNCTION_BLOCK FB_DigitalOutput IMPLEMENTS I_DigitalChannel
VAR_INPUT
END_VAR
VAR_OUTPUT
END_VAR
VAR
	sIdentifier:				STRING(25);		// Equipment ID
	Channel			AT%Q*: BOOL;	// Link to output
END_VAR

// https://github.com/PeterZerlauth/Tc3_Component

PROPERTY PUBLIC P_Identifier : STRING(25)
GET
P_Identifier:= sIdentifier;
END_GET
END_PROPERTY

PROPERTY P_State : EPlcMappingStatus
GET
P_State:= F_GetMappingStatus(adr(Channel), sizeof(BOOL));
END_GET
END_PROPERTY

PROPERTY PUBLIC P_Value : bool
GET
P_Value:= Channel;
END_GET
SET
PUBLIC 
VAR
END_VAR
Channel:= P_Value;
END_SET
END_PROPERTY

END_FUNCTION_BLOCK

// Utils/File/I_File
INTERFACE I_File

METHOD PUBLIC M_Append : BOOL
VAR_INPUT
	sText:			STRING(255);
END_VAR
END_METHOD

METHOD PUBLIC M_AppendLine : BOOL
VAR_INPUT
	sText:			STRING(255);
END_VAR
END_METHOD

METHOD PUBLIC M_Close : BOOL
VAR_INPUT
END_VAR
END_METHOD

METHOD PUBLIC M_Create : BOOL
VAR_INPUT
	sPathName:		T_MaxString;
END_VAR
END_METHOD

METHOD PUBLIC M_Delete : BOOL
VAR_INPUT
	sPathName:		T_MaxString;
END_VAR
END_METHOD

METHOD PUBLIC M_Load : BOOL
VAR_INPUT
	sPathName:		T_MaxString;
	pData:			PVOID;
	nData:			UDINT;
END_VAR
END_METHOD

METHOD PUBLIC M_Open : BOOL
VAR_INPUT
	sPathName:		T_MaxString;
END_VAR
END_METHOD

METHOD PUBLIC M_Read : BOOL
VAR_INPUT
	Value:		ANY;
END_VAR
END_METHOD

METHOD PUBLIC M_Write : BOOL
VAR_INPUT
	Value:		ANY;
END_VAR
END_METHOD

PROPERTY PUBLIC P_Error : UDINT
GET
END_GET
END_PROPERTY

END_INTERFACE
